FUNCTION_BLOCK COE_Auswertung
VAR_INPUT
END_VAR
VAR_OUTPUT
END_VAR
VAR
	MotorstromAchse1: FB_EcCoESdoRead;	
	MotorspannungAchse1: FB_EcCoESdoRead;
	MotorstromAchse2: FB_EcCoESdoRead;
	MotorspannungAchse2: FB_EcCoESdoRead;
	MotorspannungAchse3: FB_EcCoESdoRead;
	MotorstromAchse3: FB_EcCoESdoRead;
	
	Achse1Geschwindigkeit: INT;
	Achse2Geschwindigkeit: INT;
	Achse3Geschwindigkeit: INT;
	
	Achse1Motorstrom: INT;
	Achse2Motorstrom: INT;
	Achse3Motorstrom: INT;
	
	trigger: BOOL;
END_VAR

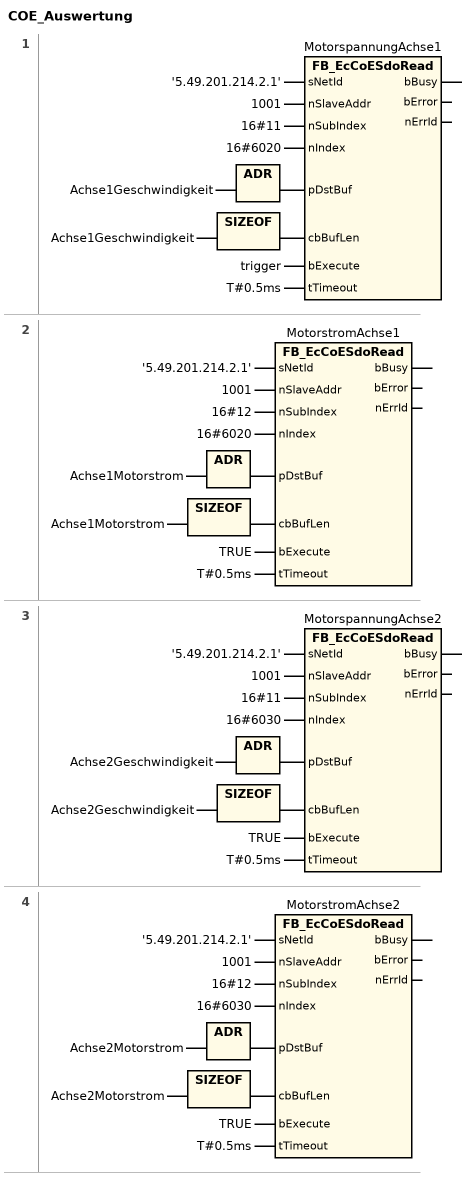
// NETWORK 1
MotorspannungAchse1(
    sNetId := '5.49.201.214.2.1',
    nSlaveAddr := 1001,
    nSubIndex := 16#11,
    nIndex := 16#6020,
    pDstBuf := ADR(Achse1Geschwindigkeit),
    cbBufLen := SIZEOF(Achse1Geschwindigkeit),
    bExecute := trigger,
    tTimeout := T#0.5ms); // FB_EcCoESdoRead

// NETWORK 2
MotorstromAchse1(
    sNetId := '5.49.201.214.2.1',
    nSlaveAddr := 1001,
    nSubIndex := 16#12,
    nIndex := 16#6020,
    pDstBuf := ADR(Achse1Motorstrom),
    cbBufLen := SIZEOF(Achse1Motorstrom),
    bExecute := TRUE,
    tTimeout := T#0.5ms); // FB_EcCoESdoRead

// NETWORK 3
MotorspannungAchse2(
    sNetId := '5.49.201.214.2.1',
    nSlaveAddr := 1001,
    nSubIndex := 16#11,
    nIndex := 16#6030,
    pDstBuf := ADR(Achse2Geschwindigkeit),
    cbBufLen := SIZEOF(Achse2Geschwindigkeit),
    bExecute := TRUE,
    tTimeout := T#0.5ms); // FB_EcCoESdoRead

// NETWORK 4
MotorstromAchse2(
    sNetId := '5.49.201.214.2.1',
    nSlaveAddr := 1001,
    nSubIndex := 16#12,
    nIndex := 16#6030,
    pDstBuf := ADR(Achse2Motorstrom),
    cbBufLen := SIZEOF(Achse2Motorstrom),
    bExecute := TRUE,
    tTimeout := T#0.5ms); // FB_EcCoESdoRead

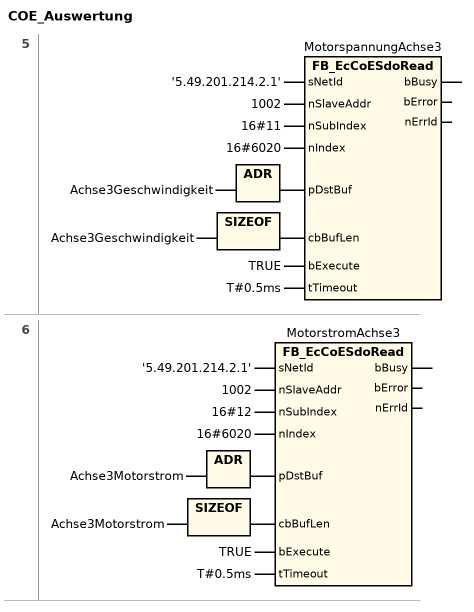
// NETWORK 5
MotorspannungAchse3(
    sNetId := '5.49.201.214.2.1',
    nSlaveAddr := 1002,
    nSubIndex := 16#11,
    nIndex := 16#6020,
    pDstBuf := ADR(Achse3Geschwindigkeit),
    cbBufLen := SIZEOF(Achse3Geschwindigkeit),
    bExecute := TRUE,
    tTimeout := T#0.5ms); // FB_EcCoESdoRead

// NETWORK 6
MotorstromAchse3(
    sNetId := '5.49.201.214.2.1',
    nSlaveAddr := 1002,
    nSubIndex := 16#12,
    nIndex := 16#6020,
    pDstBuf := ADR(Achse3Motorstrom),
    cbBufLen := SIZEOF(Achse3Motorstrom),
    bExecute := TRUE,
    tTimeout := T#0.5ms); // FB_EcCoESdoRead

END_FUNCTION_BLOCK

(* stored: Version 1.1.0.1, ProductVersion 3.1.4020.12
   POU COE_Auswertung: Id {db92f199-2295-40f9-97d2-319ddc0272f8}, SpecialFunc None *)
